{attribute addProperty BoxType "EK1122-0000-0018"}
{attribute addProperty Id "Beckhoff_EM2xxxsub_EK1100EK1100_179A0949162"}
{attribute addProperty CRC "642578266"}
{attribute addProperty SizeInBites "16"}
{attribute addProperty SizeInBytes "2"}
TYPE Beckhoff_EM2xxxEK1122_264CF75A EXTENDS EK1122_179A0949 :
STRUCT
	{attribute addProperty Name "Beckhoff_EM2xxxsub_EK1100"}
	Beckhoff_EM2xxxsub_EK1100 : EK1100_179A0949;
END_STRUCT
END_TYPE

(* stored: Version 1.2.0.0, ProductVersion 3.1.4024.9
   DUT Beckhoff_EM2xxxEK1122_264CF75A: Id {70cba534-acb3-4f81-9140-e2445f1f52d8} *)
